Universal Robots PolyScope program: changement battery.urp

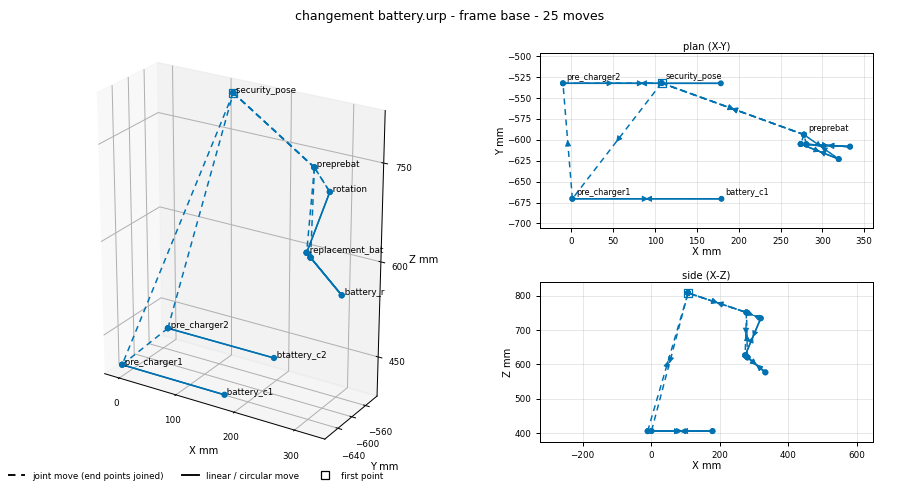
[picture p0: tool path of changement battery.urp in frame base, 25 of 25 moves have a stored position in this frame; points joined in program order, loops and branches not executed]
Program changement battery (installation=default directory=/programs/usbdisk/delete createdIn=5.11.9.1010452 lastSavedIn=5.11.9.1010452 robotSerialNumber=20225500255)
Calibrated DH parameters: a=[0.000192, -0.391659, -0.392271, 0.000079, 0.000026, 0]; d=[0.162782, -270.451826, 271.803383, -1.217811, 0.099828, 0.099665]; alpha=[1.571101, 0.000612, 0.00655, 1.570147, -1.570697, 0]; deltaTheta=[0, -0.399864, 6.705617, -0.022561, 0, 0]
Robot Program (runOnlyOnce=false)
  URCap Gripper Activate (Robotiq_Grippers, Robotiq Inc.) dataModel(ResetAndActivateKey=false)
  URCap Gripper (Robotiq_Grippers, Robotiq Inc.) dataModel(position=0.0, force=0.0, speed=0.0, positionInDouble=0.0, forceInDouble=0.0, speedInDouble=0.0, slaveIds=[9], blocking=true)
  MoveJ speed 60 deg/s, acceleration 80 deg/s^2 (useActiveTCP=true) feature=Base
    Waypoint security_pose: TCP in base x=107.72 y=-532.095 z=808.496 mm, rx=1.195 ry=1.3323 rz=1.27 rad; joints [60.184, -35.538, -17.761, -131.429, 36.815, 183.976] deg; TCP offset x=0 y=0 z=178.5 mm, rx=0 ry=0 rz=0 rad
    Waypoint preprebat: TCP in base x=278.076 y=-593.783 z=751.566 mm, rx=1.2336 ry=1.1156 rz=1.1401 rad; joints [76.407, -14.91, -57.899, -95.084, 8.153, 167.744] deg; TCP offset x=0 y=0 z=178.5 mm, rx=0 ry=0 rz=0 rad
    Waypoint replacement_bat: TCP in base x=274.085 y=-605.055 z=626.517 mm, rx=1.695 ry=1.6851 rz=0.7476 rad; joints [82.997, -46.465, -14.747, -23.656, -39.991, 80.604] deg
  MoveL speed 50 mm/s, acceleration 600 mm/s^2 (useActiveTCP=true) feature=Base
    Waypoint pre_battery: TCP in base x=280.749 y=-605.415 z=620.88 mm, rx=1.6951 ry=1.685 rz=0.7477 rad; joints [83.651, -43.843, -19.481, -22.308, -39.948, 81.616] deg
    Waypoint battery_r: TCP in base x=333.09 y=-608.135 z=576.955 mm, rx=1.695 ry=1.685 rz=0.7475 rad; joints [88.747, -31.208, -39.453, -21.046, -39.862, 89.539] deg
    URCap Gripper (Robotiq_Grippers, Robotiq Inc.) dataModel(position=100.0, force=100.0, speed=100.0, positionInDouble=100.0, forceInDouble=100.0, speedInDouble=100.0, slaveIds=[9], blocking=true)
    Waypoint pre_battery: TCP in base x=280.749 y=-605.415 z=620.88 mm, rx=1.6951 ry=1.685 rz=0.7477 rad; joints [83.651, -43.843, -19.481, -22.308, -39.948, 81.616] deg
    Waypoint replacement_bat: TCP in base x=274.085 y=-605.055 z=626.517 mm, rx=1.695 ry=1.6851 rz=0.7476 rad; joints [82.997, -46.465, -14.747, -23.656, -39.991, 80.604] deg
    Waypoint rotation: TCP in base x=319.578 y=-622.997 z=734.591 mm, rx=1.4137 ry=1.3636 rz=0.9443 rad; joints [82.267, -51.093, -5.875, -27.049, -15.913, 79.5] deg
    MoveJ speed 30 deg/s, acceleration 40 deg/s^2 (useActiveTCP=true) feature=Base
      Waypoint preprebat: TCP in base x=278.076 y=-593.783 z=751.566 mm, rx=1.2336 ry=1.1156 rz=1.1401 rad; joints [76.407, -14.91, -57.899, -95.084, 8.153, 167.744] deg
      Waypoint security_pose: TCP in base x=107.72 y=-532.095 z=808.496 mm, rx=1.195 ry=1.3323 rz=1.27 rad; joints [60.184, -35.538, -17.761, -131.429, 36.815, 183.976] deg; TCP offset x=0 y=0 z=178.5 mm, rx=0 ry=0 rz=0 rad
      Waypoint pre_charger1: TCP in base x=1.093 y=-670.444 z=406.002 mm, rx=-1.1895 ry=1.1572 rz=-1.2164 rad; joints [57.161, 16.306, -56.155, -135.023, 34.508, -4.706] deg; TCP offset x=0 y=0 z=178.5 mm, rx=0 ry=0 rz=0 rad
      MoveL speed 250 mm/s, acceleration 1200 mm/s^2 (useActiveTCP=true) feature=Base
        Waypoint battery_c1: TCP in base x=179.347 y=-670.511 z=405.98 mm, rx=-1.1892 ry=1.1573 rz=-1.2164 rad; joints [70.385, 22.04, -70.139, -123.888, 21.392, -7.843] deg
        URCap Gripper (Robotiq_Grippers, Robotiq Inc.) dataModel(position=0.0, force=100.0, speed=100.0, positionInDouble=0.0, forceInDouble=100.0, speedInDouble=100.0, slaveIds=[9], blocking=true)
        Waypoint pre_charger1: TCP in base x=1.093 y=-670.444 z=406.002 mm, rx=-1.1895 ry=1.1572 rz=-1.2164 rad; joints [57.161, 16.306, -56.155, -135.023, 34.508, -4.706] deg
        MoveJ speed 60 deg/s, acceleration 80 deg/s^2 (useActiveTCP=true) feature=Base
          Waypoint pre_charger2: TCP in base x=-10.152 y=-532.372 z=405.475 mm, rx=-1.1822 ry=1.1686 rz=-1.2283 rad; joints [48.875, 28.18, -85.963, -118.009, 41.923, -3.59] deg
          MoveL speed 250 mm/s, acceleration 1200 mm/s^2 (useActiveTCP=true) feature=Base
            Waypoint btattery_c2: TCP in base x=178.612 y=-532.417 z=405.458 mm, rx=-1.1821 ry=1.1688 rz=-1.2284 rad; joints [65.163, 32.521, -99.078, -106.95, 25.714, -6.213] deg
            URCap Gripper (Robotiq_Grippers, Robotiq Inc.) dataModel(position=100.0, force=100.0, speed=100.0, positionInDouble=100.0, forceInDouble=100.0, speedInDouble=100.0, slaveIds=[9], blocking=true)
            Waypoint pre_charger2: TCP in base x=-10.152 y=-532.372 z=405.475 mm, rx=-1.1822 ry=1.1686 rz=-1.2283 rad; joints [48.875, 28.18, -85.963, -118.009, 41.923, -3.59] deg
            MoveJ speed 60 deg/s, acceleration 80 deg/s^2 (useActiveTCP=true) feature=Base
              Waypoint security_pose: TCP in base x=107.72 y=-532.095 z=808.496 mm, rx=1.195 ry=1.3323 rz=1.27 rad; joints [60.184, -35.538, -17.761, -131.429, 36.815, 183.976] deg; TCP offset x=0 y=0 z=178.5 mm, rx=0 ry=0 rz=0 rad
              Waypoint preprebat: TCP in base x=278.076 y=-593.783 z=751.566 mm, rx=1.2336 ry=1.1156 rz=1.1401 rad; joints [76.407, -14.91, -57.899, -95.084, 8.153, 167.744] deg; TCP offset x=0 y=0 z=178.5 mm, rx=0 ry=0 rz=0 rad
              Waypoint rotation: TCP in base x=319.578 y=-622.997 z=734.591 mm, rx=1.4137 ry=1.3636 rz=0.9443 rad; joints [82.267, -51.093, -5.875, -27.049, -15.913, 79.5] deg
              MoveL speed 120 mm/s, acceleration 600 mm/s^2 (useActiveTCP=true) feature=Base
                Waypoint replacement_bat: TCP in base x=274.085 y=-605.055 z=626.517 mm, rx=1.695 ry=1.6851 rz=0.7476 rad; joints [82.997, -46.465, -14.747, -23.656, -39.991, 80.604] deg
                Waypoint pre_battery: TCP in base x=280.749 y=-605.415 z=620.88 mm, rx=1.6951 ry=1.685 rz=0.7477 rad; joints [83.651, -43.843, -19.481, -22.308, -39.948, 81.616] deg
                Waypoint battery_r: TCP in base x=333.09 y=-608.135 z=576.955 mm, rx=1.695 ry=1.685 rz=0.7475 rad; joints [88.747, -31.208, -39.453, -21.046, -39.862, 89.539] deg
                URCap Gripper (Robotiq_Grippers, Robotiq Inc.) dataModel(position=0.0, force=100.0, speed=100.0, positionInDouble=0.0, forceInDouble=100.0, speedInDouble=100.0, slaveIds=[9], blocking=true)
                Waypoint pre_battery: TCP in base x=280.749 y=-605.415 z=620.88 mm, rx=1.6951 ry=1.685 rz=0.7477 rad; joints [83.651, -43.843, -19.481, -22.308, -39.948, 81.616] deg
                MoveJ speed 60 deg/s, acceleration 80 deg/s^2 (useActiveTCP=true) feature=Base
                  Waypoint preprebat: TCP in base x=278.076 y=-593.783 z=751.566 mm, rx=1.2336 ry=1.1156 rz=1.1401 rad; joints [76.407, -14.91, -57.899, -95.084, 8.153, 167.744] deg
                  Waypoint security_pose: TCP in base x=107.72 y=-532.095 z=808.496 mm, rx=1.195 ry=1.3323 rz=1.27 rad; joints [60.184, -35.538, -17.761, -131.429, 36.815, 183.976] deg; TCP offset x=0 y=0 z=178.5 mm, rx=0 ry=0 rz=0 rad
